{attribute 'qualified_only'}
{attribute 'strict'}
TYPE ST_LaudaActualValuesCollection :
STRUCT
	BathTemperature		: REAL;
	TemperatureSetpoint	: REAL;
	PumpStage			: UINT;
	StandBy				: BOOL;
	LiquidLevel			: UINT;
END_STRUCT
END_TYPE

(* stored: Version 1.1.0.1, ProductVersion 3.1.4024.13
   DUT ST_LaudaActualValuesCollection: Id {987885e7-7ef4-0a25-34a9-b7403a66b590} *)
